Fanuc KAREL source: STR_LEN.kl

PROGRAM T
%NOLOCKGROUP
VAR
 v0 : STRING[40]
 res : INTEGER
BEGIN
 res = STR_LEN(v0)
END T
